// TIA Portal project "3 Motor 2 Anahtar Uygulaması" (V18)

(* hardware
DEVICE "S7-1200 station_1"  S7-1200 Station
   slot 0: "Rack_0"  S7-1200 Rack  Rack  V1.0
   slot 1: "PLC_1"  CPU 1214C AC/DC/Rly  6ES7 214-1BG40-0XB0  V4.6
*)

// ===== PLC "PLC_1"  CPU 1214C AC/DC/Rly =====

VAR_GLOBAL   // PLC tag table "Default tag table"
   "Stop" AT %I0.0 : Bool;
   "Start_1" AT %I0.1 : Bool;
   "Start_2" AT %I0.2 : Bool;
   "Motor_1" AT %Q0.0 : Bool;
   "Start_3" AT %I0.3 : Bool;
   "Motor_2" AT %Q0.1 : Bool;
   "Motor_3" AT %Q0.2 : Bool;
   "Aşırı Akım Koruma" AT %I0.7 : Bool;
   "Tag_1" AT %Q0.3 : Bool;
END_VAR

ORGANIZATION_BLOCK "Main"   // OB1, LAD, ProgramCycle
TITLE = "Main Program Sweep (Cycle)"
{ S7_Optimized_Access := 'TRUE' }
VERSION : 0.1
   VAR_INPUT
      Initial_Call : Bool;   // Initial call of this OB
      Remanence : Bool;   // =True, if remanent data are available
   END_VAR
BEGIN

REGION Network 1
   // *Bir sistemde 3 adet motor çalıştırılacaktır. 
   // *Sistemi çalıştırmak için 2 start ve 1 stop butonu kullanılacaktır. 
   // *1. start butonuna basıldığında 1. ve 2. motorlar çalışmaya başlayacak, 1. start butonundan el
   // çekildiğinde 1. motor duracak 2. motor çalışmaya devam edecektir.
   // *2. start butonuna basıldığında ise sadece 3. motor çalışacak, ancak 2. Motor çalışmadan 2.start butonuna basılsa bile 3. motoru çalıştırmak mümkün olmayacaktır.
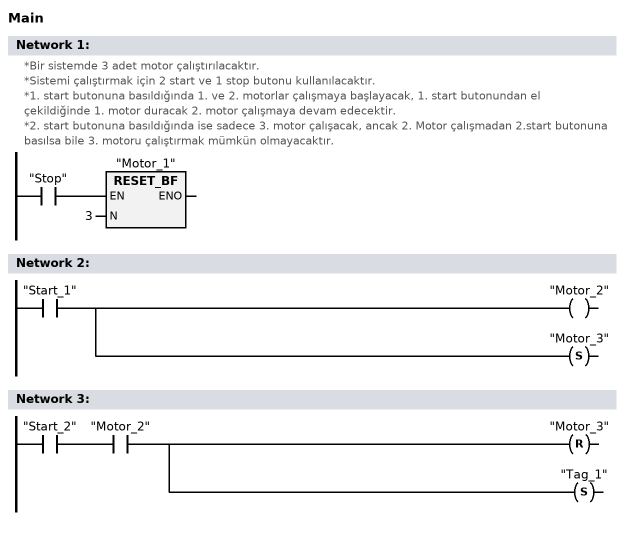
   // no SCL statement known for RBitfield: written as a call
   IF "Stop" THEN RESET_BF(operand := "Motor_1", n := 3); END_IF;
END_REGION

REGION Network 2
   RUNG wire#powerrail
      Contact( "Start_1" )
      wire#w1
      Coil( "Motor_2" )
   END_RUNG
   RUNG wire#w1
      S_Coil( "Motor_3" )
   END_RUNG
   // the same network as SCL:
   "Motor_2" := "Start_1";
   IF "Start_1" THEN "Motor_3" := TRUE; END_IF;
END_REGION

REGION Network 3
   RUNG wire#powerrail
      Contact( "Start_2" )
      Contact( "Motor_2" )
      wire#w1
      R_Coil( "Motor_3" )
   END_RUNG
   RUNG wire#w1
      S_Coil( "Tag_1" )
   END_RUNG
   // the same network as SCL:
   IF "Start_2" AND "Motor_2" THEN
       "Motor_3" := FALSE;
       "Tag_1" := TRUE;
   END_IF;
END_REGION
END_ORGANIZATION_BLOCK